(* CoDeSys 2.3.9.28 project: VISUALIZACIONBOTELLAS.pro *)
(* Libraries: Standard.lib 4.10.05 13:14:46, IecSfc.lib 13.4.06 16:51:28, SYSLIBCALLBACK.LIB 26.9.08 17:43:52 *)

(* Global variable list: Global_Variables *)
VAR_GLOBAL
   MATRIZ: ARRAY [1..5,1..10] OF REAL:=10(0),10(0),10(0),10(0),10(0);
   TIPO: ARRAY [1..10] OF INT:=1,2,2,1,1,2,2,1,1,2;
   C1:BOOL;
   C2:BOOL;
  C3:BOOL;
  C4:BOOL;
   AG:BOOL;
   LLENAR_AGUA:BOOL;
   ETIQUETAR:BOOL;
   NIVELAGUA:REAL;
   LTH:BOOL;
   LTL:BOOL;
   S2:BOOL;
   S3:BOOL;
   S4:BOOL;
  S5:BOOL;
  S6:BOOL;
   S7:BOOL;
   S8:BOOL;
   Sup1:BOOL;
   Inf1:BOOL;
	Sup2:BOOL;
   Inf2:BOOL;
   TIPO1:BOOL;
   TIPO2:BOOL;
   LLENAR:BOOL;
   LLENARTANQUE:BOOL;
   ESTIRATAP1:BOOL;
   RETRAETAP1:BOOL;
	PISTONC3:REAL;
	ESTIRATAP2:BOOL;
   RETRAETAP2:BOOL;
	PISTONC4:REAL;
   TAPONAR1:BOOL;
   TAPONAR2:BOOL;
   (*botones*)
   BOTONC1:BOOL;
   BOTONC2:BOOL;
	BOTONC3:BOOL;
   BOTONC4:BOOL;
   BOTONLLENAR:BOOL;
   BOTONLLENARTANQUE:BOOL;
  BOTONAG:BOOL;
 BOTONESTIRAPISTON3:BOOL;
	BOTONRETRAEPISTON3:BOOL;
	BOTONESTIRAPISTON4:BOOL;
	BOTONRETRAEPISTON4:BOOL;
	BOTONTAPONAR1:BOOL;
	BOTONTAPONAR2:BOOL;
(*VARIABLES MODO OPERACIÓN*)
    MANUAL:BOOL;
    AUTO:BOOL;
    C2OCUP:BOOL;
    TANQUELLENANDO:BOOL;
    TANQUEVACIO:BOOL;
    M:BOOL;
    PARO:BOOL;
    MARCHA:BOOL;
    MODORESET:BOOL;
(*variables temporizadores*)
    AT2:BOOL;
    FT2:BOOL;
    AT1:BOOL;
    FT1:BOOL;
    AT3:BOOL;
    FT3:BOOL;
  	AT4:BOOL;
    FT4:BOOL;
    Vectorcola:ARRAY [1..11] OF INT;
    ACCOMPLISHED:BOOL;
	TAPONADORA2OCU:BOOL;
    TAPONADORA1OCU:BOOL;
    RESETC3:BOOL;
    RESETC4:BOOL;
(*variables creadas*)
	C2OCU: BOOL;
	DEPOSOCU: BOOL;
	FLANCOS2SUBIDA: BOOL;
	FLANCOS4SUBIDA: BOOL;
	FLANCOS5SUBIDA: BOOL;
	FLANCOS7BAJADA: BOOL;
	FLANCOS34BAJADA: BOOL;
	FLANCOS8BAJADA: BOOL;
	TAP1OCU: BOOL;
	TAP2OCU: BOOL;
	CONTROLTANQUE: BOOL;
	AT30: BOOL;
	FT30: BOOL;

END_VAR

(* POU PLC_PRG, ST *)
PROGRAM PLC_PRG
VAR
END_VAR
VISUALIZACION;
MODOS;
TEMPOYCONTA;
END_PROGRAM

(* POU VISUALIZACION, ST *)
PROGRAM VISUALIZACION
VAR
	T1:TON;
	TH_OUT: BOOL;
    I:INT;
	RETRAETAP1THEN: BOOL;
END_VAR
AUTO:=NOT MANUAL;

T1(IN:=C1 AND NOT TH_OUT,PT:=T#4s,Q=>TH_OUT);
(*HACER VISIBLES BOTELLAS*)

IF C1=TRUE AND TH_OUT=TRUE AND MODORESET=FALSE THEN
   FOR I:=1 TO 10 BY 1 DO
      IF MATRIZ[1,I]=0 THEN
        MATRIZ[1,I]:=1;
        EXIT;
	  END_IF;
   END_FOR;
END_IF;

(*MOVIMIENTO BOTELLAS, PRIMER TRAMO HASTA 590*)
FOR I:=1 TO 10 BY 1 DO
   IF C1=TRUE AND MATRIZ[1,I]=1 AND MATRIZ[2,I]<590  THEN
     IF MODORESET=FALSE THEN
      MATRIZ[2,I]:=MATRIZ[2,I]+2;
    ELSE
       IF MATRIZ[2,I]>1 THEN
            MATRIZ[2,I]:=MATRIZ[2,I]+2;
      END_IF;
    END_IF;
   END_IF;
END_FOR;

(*LLENAR BOTELLAS*)

FOR I:=1 TO 10 BY 1 DO
	IF MATRIZ[2,I]>419 AND MATRIZ[2,I]<431 AND LLENAR=TRUE AND MATRIZ[5,I]=0 THEN
  	 MATRIZ[5,I]:=1;
	EXIT;
	END_IF;
END_FOR;
(*MOVIMIENTO EN LA SEGUNDA CINTA*)
FOR I:=1 TO 10 BY 1 DO
   IF C2=TRUE AND MATRIZ[1,I]=1 AND MATRIZ[2,I]>=575 AND MATRIZ[2,I]<730 AND AG=1 THEN
      MATRIZ[2,I]:=MATRIZ[2,I]+4;
      MATRIZ[3,I]:=MATRIZ[3,I]-4;
       IF MATRIZ[3,I]<=-130 THEN

         MATRIZ[3,I]:=-130;
       END_IF;
   END_IF;
IF C2=TRUE AND MATRIZ[1,I]=1 AND MATRIZ[2,I]>=575 AND MATRIZ[2,I]<734  AND AG=0 THEN
      MATRIZ[2,I]:=MATRIZ[2,I]+4;
      MATRIZ[3,I]:=MATRIZ[3,I]+4;
       IF MATRIZ[3,I]>=140 THEN
           MATRIZ[3,I]:=140;
      END_IF;
   END_IF;
END_FOR;

(*CINTA3*)
FOR I:=1 TO 10 BY 1 DO
   IF C3=TRUE AND MATRIZ[1,I]=1 AND MATRIZ[2,I]>=730 AND MATRIZ[3,I]<0 THEN
        MATRIZ[2,I]:=MATRIZ[2,I]+2;

       END_IF;
END_FOR;

(*CINTA3*)
FOR I:=1 TO 10 BY 1 DO
   IF C4=TRUE AND MATRIZ[1,I]=1 AND MATRIZ[2,I]>=730 AND MATRIZ[3,I]>0 THEN
        MATRIZ[2,I]:=MATRIZ[2,I]+2;
   END_IF;
END_FOR;

(*TANQUE*)
IF LLENAR=TRUE THEN
 NIVELAGUA:=NIVELAGUA+1;
 IF NIVELAGUA>198 THEN
     NIVELAGUA:=198;
 END_IF;
END_IF

IF LLENARTANQUE=TRUE THEN
 NIVELAGUA:=NIVELAGUA-2;
 IF NIVELAGUA<=0 THEN
     NIVELAGUA:=0;
 END_IF;
END_IF

(*PISTON TAPONADORA 1*)
IF ESTIRATAP1 THEN
PISTONC3:=PISTONC3+3;
      IF PISTONC3>=+30 THEN
           PISTONC3:=+30;
     END_IF;

END_IF;
IF RETRAETAP1 THEN
      PISTONC3:=PISTONC3-3;
      IF PISTONC3<=0 THEN
           PISTONC3:=0;
     END_IF;
END_IF;

(*PISTON TAPONADORA 2*)
IF ESTIRATAP2 THEN
PISTONC4:=PISTONC4+3;
      IF PISTONC4>=+40 THEN
           PISTONC4:=+40;
     END_IF;

END_IF;
IF RETRAETAP2 THEN
      PISTONC4:=PISTONC4-3;
      IF PISTONC4<=0 THEN
           PISTONC4:=0;
     END_IF;
END_IF;

(*SENSORES*)
FOR I:=1 TO 10 BY 1 DO
   IF MATRIZ[2,I]>419 AND MATRIZ[2,I]<431 AND TIPO[I]=1 THEN
         TIPO1:=TRUE;
         EXIT;
   ELSE
         TIPO1:=FALSE;
   END_IF;
   IF MATRIZ[2,I]>419 AND MATRIZ[2,I]<431 AND TIPO[I]=2 THEN
         TIPO2:=TRUE;
         EXIT;
   ELSE
         TIPO2:=FALSE;
   END_IF;
END_FOR;


FOR I:=1 TO 10 BY 1 DO
   IF MATRIZ[2,I]>570 AND MATRIZ[2,I]<600 THEN
         S2:=TRUE;
         EXIT;
   ELSE
         S2:=FALSE;
   END_IF;
END_FOR;

IF NIVELAGUA<2 THEN
    LTH:=TRUE;
ELSE
    LTH:=FALSE;
END_IF;

IF NIVELAGUA<90 THEN
    LTL:=TRUE;
ELSE
    LTL:=FALSE;
END_IF;

FOR I:=1 TO 10 BY 1 DO
   IF MATRIZ[2,I]>733 AND MATRIZ[2,I]<745 AND MATRIZ[3,I]>0 THEN
         S3:=TRUE;
         EXIT;
   ELSE
         S3:=FALSE;
   END_IF;
END_FOR;


FOR I:=1 TO 10 BY 1 DO
   IF MATRIZ[2,I]>729 AND MATRIZ[2,I]<745 AND MATRIZ[3,I] <0 THEN
         S4:=TRUE;
         EXIT;
   ELSE
         S4:=FALSE;
   END_IF;
END_FOR;

FOR I:=1 TO 10 BY 1 DO
   IF MATRIZ[2,I]>920 AND MATRIZ[2,I]<935 AND MATRIZ[3,I] <0 THEN
         S6:=TRUE;
         EXIT;
   ELSE
         S6:=FALSE;
   END_IF;
END_FOR;

FOR I:=1 TO 10 BY 1 DO
   IF MATRIZ[2,I]>1075 AND MATRIZ[2,I]<1090 AND MATRIZ[3,I] <0 THEN
         S8:=TRUE;
         EXIT;
   ELSE
         S8:=FALSE;
   END_IF;
END_FOR;


FOR I:=1 TO 10 BY 1 DO
   IF MATRIZ[2,I]>920 AND MATRIZ[2,I]<935 AND MATRIZ[3,I] >0 THEN
         S5:=TRUE;
         EXIT;
   ELSE
         S5:=FALSE;
   END_IF;
END_FOR;

FOR I:=1 TO 10 BY 1 DO
   IF MATRIZ[2,I]>1075 AND MATRIZ[2,I]<1090 AND MATRIZ[3,I] >0 THEN
         S7:=TRUE;
         EXIT;
   ELSE
         S7:=FALSE;
   END_IF;
END_FOR;
(*PISTON C3*)
IF PISTONC3=0 THEN
     Sup1:=TRUE;
ELSE
    Sup1:=FALSE;
END_IF;
IF PISTONC3>29 THEN
     Inf1:=TRUE;
ELSE
    Inf1:=FALSE;
END_IF;

(*PISTON C4*)
IF PISTONC4=0 THEN
     Sup2:=TRUE;
ELSE
    Sup2:=FALSE;
END_IF;
IF PISTONC4>39 THEN
     Inf2:=TRUE;
ELSE
    Inf2:=FALSE;
END_IF;


(*REINICIO DE TODO*)

FOR I:=1 TO 10 BY 1 DO
   IF MATRIZ[2,I]>=1089  THEN
    MATRIZ[1,I]:=0;
    MATRIZ[2,I]:=0;
    MATRIZ[3,I]:=0;
   MATRIZ[4,I]:=0;
   MATRIZ[5,I]:=0;
   END_IF;
END_FOR;
END_PROGRAM

(* POU MODOS, SFC *)
PROGRAM MODOS
VAR
	AUTOMATICO: BOOL;
END_VAR
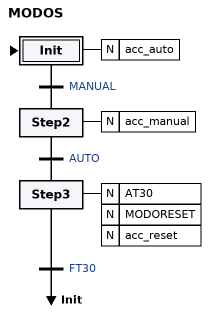
INITIAL_STEP Init:
	acc_auto(N);
END_STEP
TRANSITION FROM Init TO Step2 := MANUAL;
END_TRANSITION
STEP Step2:
	acc_manual(N);
END_STEP
TRANSITION FROM Step2 TO Step3 := AUTO;
END_TRANSITION
STEP Step3:
	AT30(N);
	MODORESET(N);
	acc_reset(N);
END_STEP
TRANSITION FROM Step3 TO Init := FT30;
END_TRANSITION
END_PROGRAM
ACTION acc_auto:
AUTOMATICO1;
END_ACTION
ACTION acc_manual:
MANUAL_PROG;
END_ACTION
ACTION acc_reset:
REINICIO;
Encolar;
Mover_cinta2;
END_ACTION

(* POU AUTOMATICO1, SFC *)
PROGRAM AUTOMATICO1
VAR
END_VAR
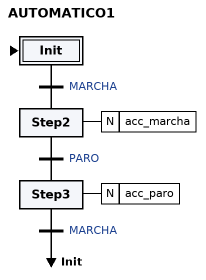
INITIAL_STEP Init:
END_STEP
TRANSITION FROM Init TO Step2 := MARCHA;
END_TRANSITION
STEP Step2:
	acc_marcha(N);
END_STEP
TRANSITION FROM Step2 TO Step3 := PARO;
END_TRANSITION
STEP Step3:
	acc_paro(N);
END_STEP
TRANSITION FROM Step3 TO Init := MARCHA;
END_TRANSITION
END_PROGRAM
ACTION acc_marcha:
Cinta1;
CINTA2;
CINTA3;
CINTA4;
Tanque1;
TANQUE2;
TAPONADOR1;
TAPONADOR2;
Encolar;
Mover_cinta2;
END_ACTION
ACTION acc_paro:
PARO1;
Tanque1;
TAPONADOR1;
TAPONADOR2;
END_ACTION

(* POU Cinta1, LD *)
PROGRAM Cinta1
VAR
END_VAR
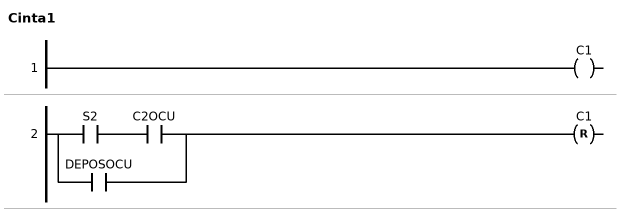
_LD_ (* Ladder Diagram *)
NETWORK 1
	* --- (C1)
NETWORK 2
	{ [S2] - [C2OCU] | [DEPOSOCU] } --- (R C1)
_END_LD_
(* the same logic as Structured Text *)
(* Network 1 *)
C1 := TRUE;
(* Network 2 *)
IF S2 AND C2OCU OR DEPOSOCU THEN C1 := FALSE; END_IF;
END_PROGRAM

(* POU PARO1, LD *)
PROGRAM PARO1
VAR
END_VAR
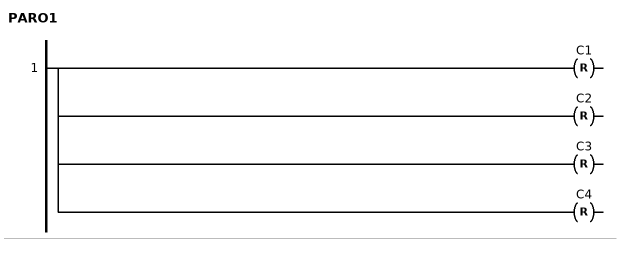
_LD_ (* Ladder Diagram *)
NETWORK 1
	* --- (R C1) (R C2) (R C3) (R C4)
_END_LD_
(* the same logic as Structured Text *)
(* Network 1 *)
C1 := FALSE;
C2 := FALSE;
C3 := FALSE;
C4 := FALSE;
END_PROGRAM

(* POU MANUAL_PROG, LD *)
PROGRAM MANUAL_PROG
VAR
END_VAR
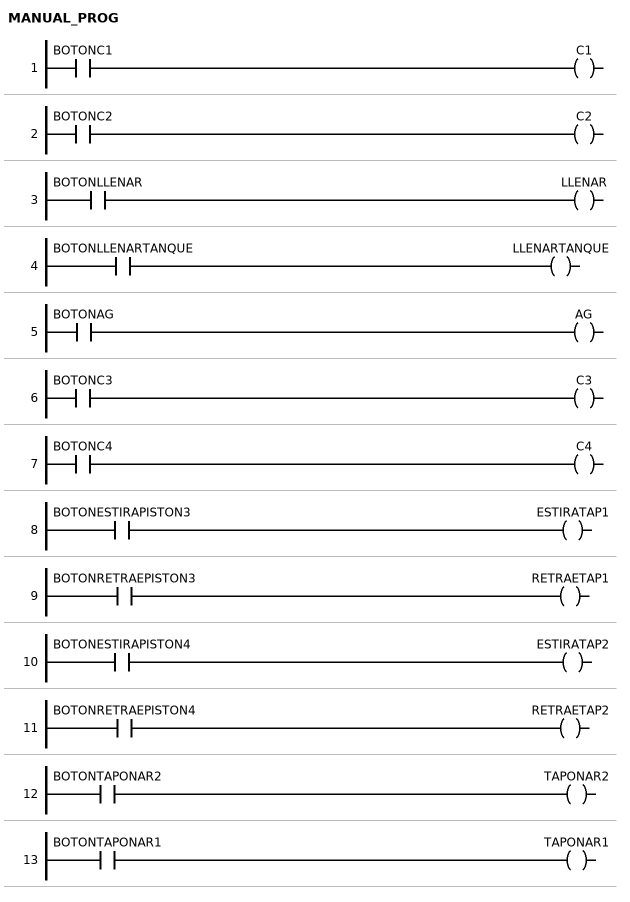
_LD_ (* Ladder Diagram *)
NETWORK 1
	[BOTONC1] --- (C1)
NETWORK 2
	[BOTONC2] --- (C2)
NETWORK 3
	[BOTONLLENAR] --- (LLENAR)
NETWORK 4
	[BOTONLLENARTANQUE] --- (LLENARTANQUE)
NETWORK 5
	[BOTONAG] --- (AG)
NETWORK 6
	[BOTONC3] --- (C3)
NETWORK 7
	[BOTONC4] --- (C4)
NETWORK 8
	[BOTONESTIRAPISTON3] --- (ESTIRATAP1)
NETWORK 9
	[BOTONRETRAEPISTON3] --- (RETRAETAP1)
NETWORK 10
	[BOTONESTIRAPISTON4] --- (ESTIRATAP2)
NETWORK 11
	[BOTONRETRAEPISTON4] --- (RETRAETAP2)
NETWORK 12
	[BOTONTAPONAR2] --- (TAPONAR2)
NETWORK 13
	[BOTONTAPONAR1] --- (TAPONAR1)
_END_LD_
(* the same logic as Structured Text *)
(* Network 1 *)
C1 := BOTONC1;
(* Network 2 *)
C2 := BOTONC2;
(* Network 3 *)
LLENAR := BOTONLLENAR;
(* Network 4 *)
LLENARTANQUE := BOTONLLENARTANQUE;
(* Network 5 *)
AG := BOTONAG;
(* Network 6 *)
C3 := BOTONC3;
(* Network 7 *)
C4 := BOTONC4;
(* Network 8 *)
ESTIRATAP1 := BOTONESTIRAPISTON3;
(* Network 9 *)
RETRAETAP1 := BOTONRETRAEPISTON3;
(* Network 10 *)
ESTIRATAP2 := BOTONESTIRAPISTON4;
(* Network 11 *)
RETRAETAP2 := BOTONRETRAEPISTON4;
(* Network 12 *)
TAPONAR2 := BOTONTAPONAR2;
(* Network 13 *)
TAPONAR1 := BOTONTAPONAR1;
END_PROGRAM

(* POU REINICIO, LD *)
PROGRAM REINICIO
VAR
END_VAR
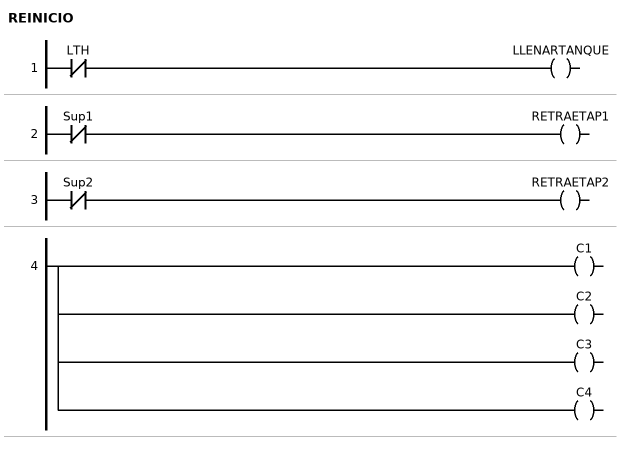
_LD_ (* Ladder Diagram *)
NETWORK 1
	[/LTH] --- (LLENARTANQUE)
NETWORK 2
	[/Sup1] --- (RETRAETAP1)
NETWORK 3
	[/Sup2] --- (RETRAETAP2)
NETWORK 4
	* --- (C1) (C2) (C3) (C4)
_END_LD_
(* the same logic as Structured Text *)
(* Network 1 *)
LLENARTANQUE := NOT LTH;
(* Network 2 *)
RETRAETAP1 := NOT Sup1;
(* Network 3 *)
RETRAETAP2 := NOT Sup2;
(* Network 4 *)
C1 := TRUE;
C2 := TRUE;
C3 := TRUE;
C4 := TRUE;
END_PROGRAM

(* POU TEMPOYCONTA, LD *)
PROGRAM TEMPOYCONTA
VAR
	T1: TON;
	T2: TON;
	T3: TON;
	T4: TON;
	T30: TON;


END_VAR
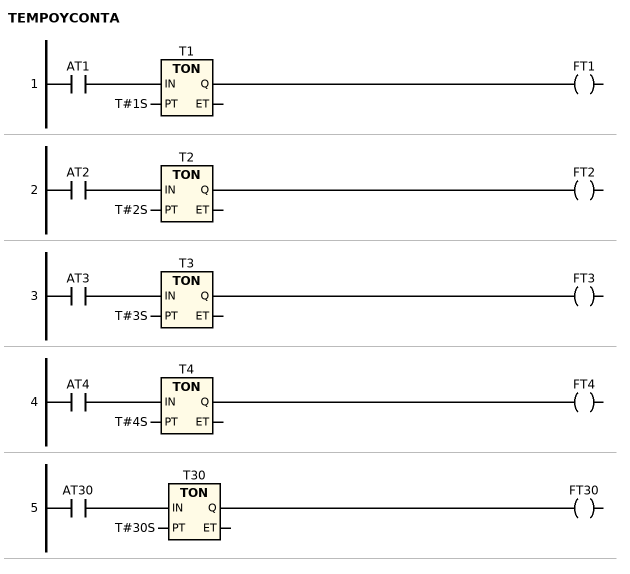
_LD_ (* Ladder Diagram *)
NETWORK 1
	[AT1] - T1:TON(IN: *, PT: T#1S) --- (FT1)
NETWORK 2
	[AT2] - T2:TON(IN: *, PT: T#2S) --- (FT2)
NETWORK 3
	[AT3] - T3:TON(IN: *, PT: T#3S) --- (FT3)
NETWORK 4
	[AT4] - T4:TON(IN: *, PT: T#4S) --- (FT4)
NETWORK 5
	[AT30] - T30:TON(IN: *, PT: T#30S) --- (FT30)
_END_LD_
(* the same logic as Structured Text *)
(* Network 1 *)
T1(IN := AT1, PT := T#1S);
FT1 := T1.Q;
(* Network 2 *)
T2(IN := AT2, PT := T#2S);
FT2 := T2.Q;
(* Network 3 *)
T3(IN := AT3, PT := T#3S);
FT3 := T3.Q;
(* Network 4 *)
T4(IN := AT4, PT := T#4S);
FT4 := T4.Q;
(* Network 5 *)
T30(IN := AT30, PT := T#30S);
FT30 := T30.Q;
END_PROGRAM

(* POU CINTA2, LD *)
PROGRAM CINTA2
VAR
	TRIG1: R_TRIG;
	TRIG2: F_TRIG;
	TRIG3: F_TRIG;
	CTUD1: CTUD;
	RESETC2: BOOL;

END_VAR
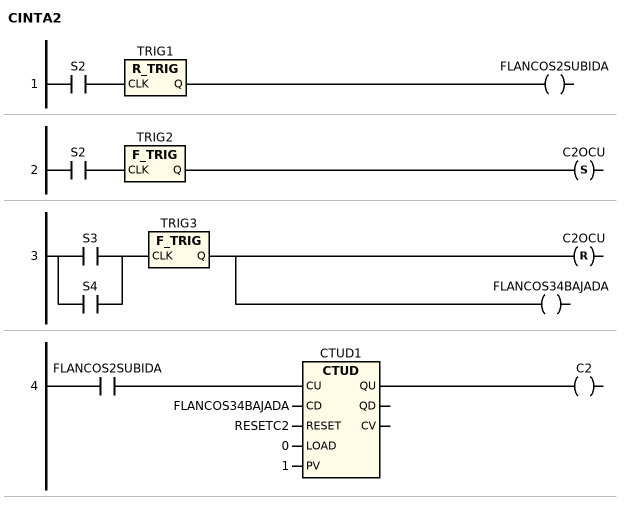
_LD_ (* Ladder Diagram *)
NETWORK 1
	[S2] - TRIG1:R_TRIG(CLK: *) --- (FLANCOS2SUBIDA)
NETWORK 2
	[S2] - TRIG2:F_TRIG(CLK: *) --- (S C2OCU)
NETWORK 3
	{ [S3] | [S4] } - TRIG3:F_TRIG(CLK: *) --- (R C2OCU) (FLANCOS34BAJADA)
NETWORK 4
	[FLANCOS2SUBIDA] - CTUD1:CTUD(CU: *, CD: FLANCOS34BAJADA, RESET: RESETC2, LOAD: 0, PV: 1) --- (C2)
_END_LD_
(* the same logic as Structured Text *)
(* Network 1 *)
TRIG1(CLK := S2);
FLANCOS2SUBIDA := TRIG1.Q;
(* Network 2 *)
TRIG2(CLK := S2);
IF TRIG2.Q THEN C2OCU := TRUE; END_IF;
(* Network 3 *)
TRIG3(CLK := S3 OR S4);
IF TRIG3.Q THEN C2OCU := FALSE; END_IF;
FLANCOS34BAJADA := TRIG3.Q;
(* Network 4 *)
CTUD1(CU := FLANCOS2SUBIDA, CD := FLANCOS34BAJADA, RESET := RESETC2, LOAD := 0, PV := 1);
C2 := CTUD1.QU;
END_PROGRAM

(* POU CINTA3, LD *)
PROGRAM CINTA3
VAR
	TRIG1: R_TRIG;
	TRIG2: F_TRIG;
    CTUD1:  CTUD;
END_VAR
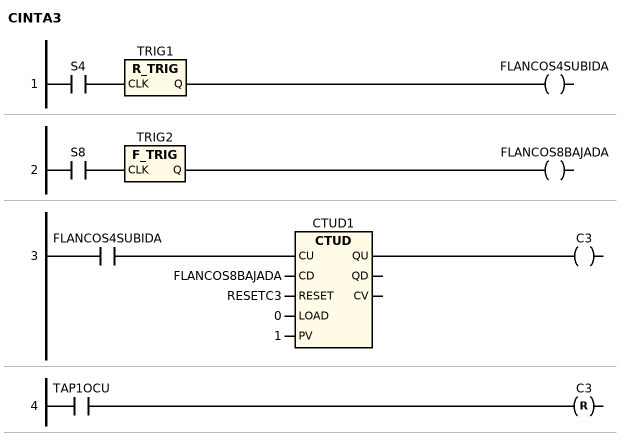
_LD_ (* Ladder Diagram *)
NETWORK 1
	[S4] - TRIG1:R_TRIG(CLK: *) --- (FLANCOS4SUBIDA)
NETWORK 2
	[S8] - TRIG2:F_TRIG(CLK: *) --- (FLANCOS8BAJADA)
NETWORK 3
	[FLANCOS4SUBIDA] - CTUD1:CTUD(CU: *, CD: FLANCOS8BAJADA, RESET: RESETC3, LOAD: 0, PV: 1) --- (C3)
NETWORK 4
	[TAP1OCU] --- (R C3)
_END_LD_
(* the same logic as Structured Text *)
(* Network 1 *)
TRIG1(CLK := S4);
FLANCOS4SUBIDA := TRIG1.Q;
(* Network 2 *)
TRIG2(CLK := S8);
FLANCOS8BAJADA := TRIG2.Q;
(* Network 3 *)
CTUD1(CU := FLANCOS4SUBIDA, CD := FLANCOS8BAJADA, RESET := RESETC3, LOAD := 0, PV := 1);
C3 := CTUD1.QU;
(* Network 4 *)
IF TAP1OCU THEN C3 := FALSE; END_IF;
END_PROGRAM

(* POU CINTA4, LD *)
PROGRAM CINTA4
VAR
	TRIG1: R_TRIG;
	TRIG2: F_TRIG;
    CTUD1:  CTUD;
END_VAR
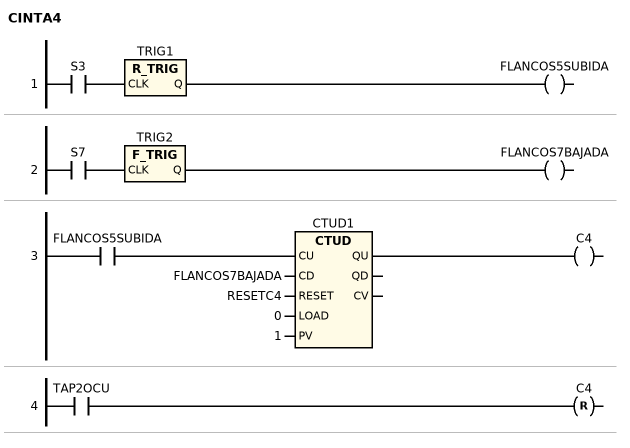
_LD_ (* Ladder Diagram *)
NETWORK 1
	[S3] - TRIG1:R_TRIG(CLK: *) --- (FLANCOS5SUBIDA)
NETWORK 2
	[S7] - TRIG2:F_TRIG(CLK: *) --- (FLANCOS7BAJADA)
NETWORK 3
	[FLANCOS5SUBIDA] - CTUD1:CTUD(CU: *, CD: FLANCOS7BAJADA, RESET: RESETC4, LOAD: 0, PV: 1) --- (C4)
NETWORK 4
	[TAP2OCU] --- (R C4)
_END_LD_
(* the same logic as Structured Text *)
(* Network 1 *)
TRIG1(CLK := S3);
FLANCOS5SUBIDA := TRIG1.Q;
(* Network 2 *)
TRIG2(CLK := S7);
FLANCOS7BAJADA := TRIG2.Q;
(* Network 3 *)
CTUD1(CU := FLANCOS5SUBIDA, CD := FLANCOS7BAJADA, RESET := RESETC4, LOAD := 0, PV := 1);
C4 := CTUD1.QU;
(* Network 4 *)
IF TAP2OCU THEN C4 := FALSE; END_IF;
END_PROGRAM

(* POU Encolar, ST *)
PROGRAM Encolar
VAR


	TIPO1a:BOOL;
    TIPO2a:BOOL;


	I: INT;

	Acca: BOOL;

END_VAR
IF TIPO1=TRUE AND TIPO1a=FALSE THEN
	FOR I:= 1 TO 10 BY 1 DO
		IF Vectorcola[I] = 0 THEN
			Vectorcola[I]:= 1;
			EXIT;
		END_IF;
	END_FOR;
END_IF;


IF TIPO2=TRUE AND TIPO2a=FALSE THEN
	FOR I:= 1 TO 10 BY 1 DO
		IF Vectorcola[I] = 0 THEN
			Vectorcola[I]:= 2;
			EXIT;
		END_IF;
	END_FOR;
END_IF;


IF ACCOMPLISHED = TRUE AND ACCa = FALSE THEN
	FOR I:=1 TO 10 BY 1 DO
		Vectorcola[I]:= Vectorcola[I+1];
	END_FOR;
		Vectorcola[10]:= 0;
	END_IF;




TIPO1a:=TIPO1;
TIPO2a:=TIPO2;
Acca:= ACCOMPLISHED;
END_PROGRAM

(* POU Mover_cinta2, SFC *)
PROGRAM Mover_cinta2
VAR
END_VAR
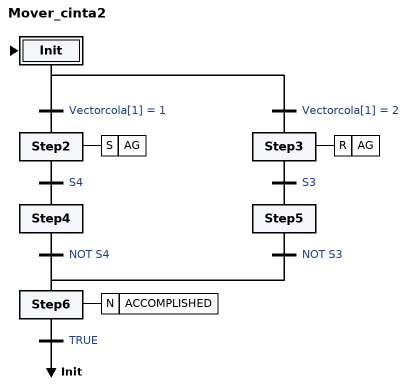
INITIAL_STEP Init:
END_STEP
TRANSITION FROM Init TO Step2 := Vectorcola[1] = 1;
END_TRANSITION
TRANSITION FROM Init TO Step3 := Vectorcola[1] = 2;
END_TRANSITION
STEP Step2:
	AG(S);
END_STEP
TRANSITION FROM Step2 TO Step4 := S4;
END_TRANSITION
STEP Step4:
END_STEP
TRANSITION FROM Step4 TO Step6 := NOT S4;
END_TRANSITION
STEP Step3:
	AG(R);
END_STEP
TRANSITION FROM Step3 TO Step5 := S3;
END_TRANSITION
STEP Step5:
END_STEP
TRANSITION FROM Step5 TO Step6 := NOT S3;
END_TRANSITION
STEP Step6:
	ACCOMPLISHED(N);
END_STEP
TRANSITION FROM Step6 TO Init := TRUE;
END_TRANSITION
END_PROGRAM

(* POU Tanque1, SFC *)
PROGRAM Tanque1
VAR
END_VAR
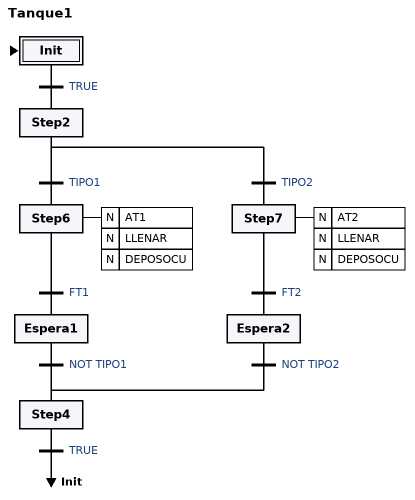
INITIAL_STEP Init:
END_STEP
TRANSITION FROM Init TO Step2 := TRUE;
END_TRANSITION
STEP Step2:
END_STEP
TRANSITION FROM Step2 TO Step6 := TIPO1;
END_TRANSITION
TRANSITION FROM Step2 TO Step7 := TIPO2;
END_TRANSITION
STEP Step6:
	AT1(N);
	LLENAR(N);
	DEPOSOCU(N);
END_STEP
TRANSITION FROM Step6 TO Espera1 := FT1;
END_TRANSITION
STEP Espera1:
END_STEP
TRANSITION FROM Espera1 TO Step4 := NOT TIPO1;
END_TRANSITION
STEP Step7:
	AT2(N);
	LLENAR(N);
	DEPOSOCU(N);
END_STEP
TRANSITION FROM Step7 TO Espera2 := FT2;
END_TRANSITION
STEP Espera2:
END_STEP
TRANSITION FROM Espera2 TO Step4 := NOT TIPO2;
END_TRANSITION
STEP Step4:
END_STEP
TRANSITION FROM Step4 TO Init := TRUE;
END_TRANSITION
END_PROGRAM

(* POU TANQUE2, LD *)
PROGRAM TANQUE2
VAR
END_VAR
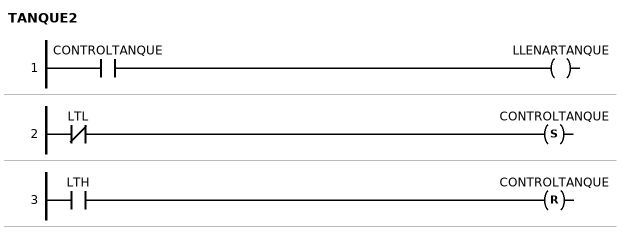
_LD_ (* Ladder Diagram *)
NETWORK 1
	[CONTROLTANQUE] --- (LLENARTANQUE)
NETWORK 2
	[/LTL] --- (S CONTROLTANQUE)
NETWORK 3
	[LTH] --- (R CONTROLTANQUE)
_END_LD_
(* the same logic as Structured Text *)
(* Network 1 *)
LLENARTANQUE := CONTROLTANQUE;
(* Network 2 *)
IF NOT LTL THEN CONTROLTANQUE := TRUE; END_IF;
(* Network 3 *)
IF LTH THEN CONTROLTANQUE := FALSE; END_IF;
END_PROGRAM

(* POU TAPONADOR1, SFC *)
PROGRAM TAPONADOR1
VAR
END_VAR
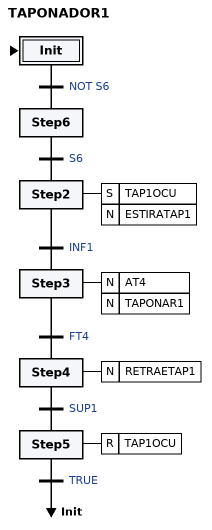
INITIAL_STEP Init:
END_STEP
TRANSITION FROM Init TO Step6 := NOT S6;
END_TRANSITION
STEP Step6:
END_STEP
TRANSITION FROM Step6 TO Step2 := S6;
END_TRANSITION
STEP Step2:
	TAP1OCU(S);
	ESTIRATAP1(N);
END_STEP
TRANSITION FROM Step2 TO Step3 := INF1;
END_TRANSITION
STEP Step3:
	AT4(N);
	TAPONAR1(N);
END_STEP
TRANSITION FROM Step3 TO Step4 := FT4;
END_TRANSITION
STEP Step4:
	RETRAETAP1(N);
END_STEP
TRANSITION FROM Step4 TO Step5 := SUP1;
END_TRANSITION
STEP Step5:
	TAP1OCU(R);
END_STEP
TRANSITION FROM Step5 TO Init := TRUE;
END_TRANSITION
END_PROGRAM

(* POU TAPONADOR2, SFC *)
PROGRAM TAPONADOR2
VAR
END_VAR
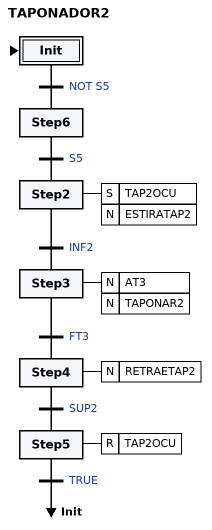
INITIAL_STEP Init:
END_STEP
TRANSITION FROM Init TO Step6 := NOT S5;
END_TRANSITION
STEP Step6:
END_STEP
TRANSITION FROM Step6 TO Step2 := S5;
END_TRANSITION
STEP Step2:
	TAP2OCU(S);
	ESTIRATAP2(N);
END_STEP
TRANSITION FROM Step2 TO Step3 := INF2;
END_TRANSITION
STEP Step3:
	AT3(N);
	TAPONAR2(N);
END_STEP
TRANSITION FROM Step3 TO Step4 := FT3;
END_TRANSITION
STEP Step4:
	RETRAETAP2(N);
END_STEP
TRANSITION FROM Step4 TO Step5 := SUP2;
END_TRANSITION
STEP Step5:
	TAP2OCU(R);
END_STEP
TRANSITION FROM Step5 TO Init := TRUE;
END_TRANSITION
END_PROGRAM

(* Visualisation VISUAL
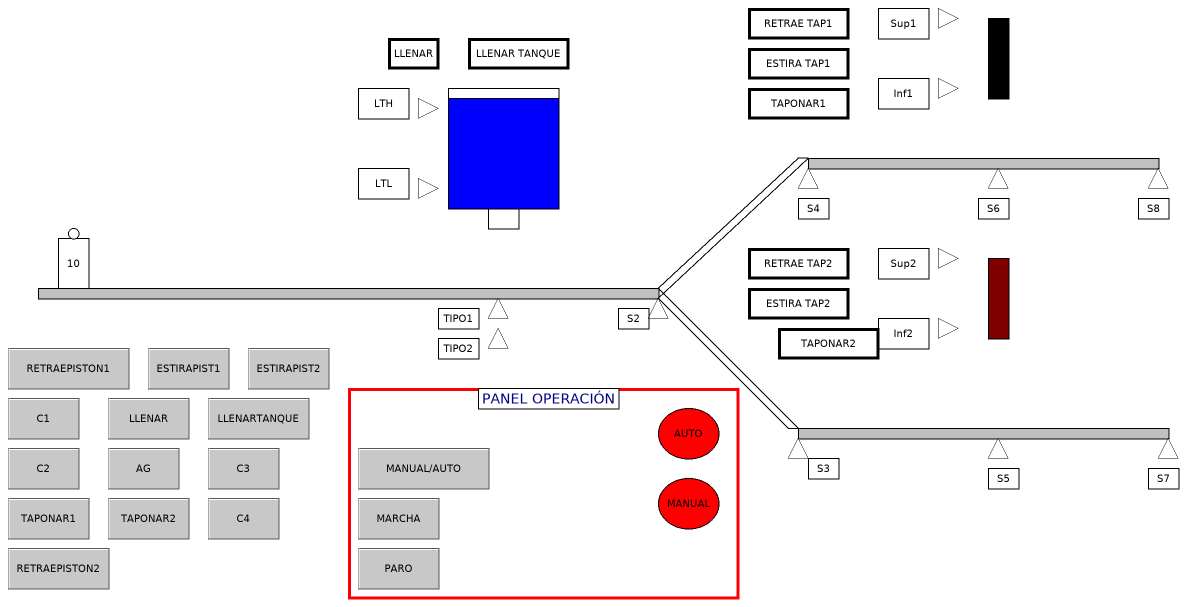
rectangle at (60,260)-(91,291): text "1"; invisible if MATRIZ[1,1]=0; alarm colour if MATRIZ[5,1]; x offset MATRIZ[2,1]; y offset MATRIZ[3,1]
ellipse at (70,250)-(81,261): invisible if MATRIZ[1,1]=0; x offset MATRIZ[2,1]; y offset MATRIZ[3,1]
rectangle at (60,240)-(91,291): text "2"; invisible if MATRIZ[1,2]=0; alarm colour if MATRIZ[5,2]; x offset MATRIZ[2,2]; y offset MATRIZ[3,2]
ellipse at (70,230)-(81,241): invisible if MATRIZ[1,2]=0; x offset MATRIZ[2,2]; y offset MATRIZ[3,2]
rectangle at (60,240)-(91,291): text "3"; invisible if MATRIZ[1,3]=0; alarm colour if MATRIZ[5,3]; x offset MATRIZ[2,3]; y offset MATRIZ[3,3]
ellipse at (70,230)-(81,241): invisible if MATRIZ[1,3]=0; x offset MATRIZ[2,3]; y offset MATRIZ[3,3]
rectangle at (60,260)-(91,291): text "4"; invisible if MATRIZ[1,4]=0; alarm colour if MATRIZ[5,4]; x offset MATRIZ[2,4]; y offset MATRIZ[3,4]
ellipse at (70,250)-(81,261): invisible if MATRIZ[1,4]=0; x offset MATRIZ[2,4]; y offset MATRIZ[3,4]
rectangle at (60,260)-(91,291): text "5"; invisible if MATRIZ[1,5]=0; alarm colour if MATRIZ[5,5]; x offset MATRIZ[2,5]; y offset MATRIZ[3,5]
ellipse at (70,250)-(81,261): invisible if MATRIZ[1,5]=0; x offset MATRIZ[2,5]; y offset MATRIZ[3,5]
rectangle at (60,240)-(91,291): text "6"; invisible if MATRIZ[1,6]=0; alarm colour if MATRIZ[5,6]; x offset MATRIZ[2,6]; y offset MATRIZ[3,6]
ellipse at (70,230)-(81,241): invisible if MATRIZ[1,6]=0; x offset MATRIZ[2,6]; y offset MATRIZ[3,6]
rectangle at (60,240)-(91,291): text "7"; invisible if MATRIZ[1,7]=0; alarm colour if MATRIZ[5,7]; x offset MATRIZ[2,7]; y offset MATRIZ[3,7]
ellipse at (70,230)-(81,241): invisible if MATRIZ[1,7]=0; x offset MATRIZ[2,7]; y offset MATRIZ[3,7]
rectangle at (60,260)-(91,291): text "8"; invisible if MATRIZ[1,8]=0; alarm colour if MATRIZ[5,8]; x offset MATRIZ[2,8]; y offset MATRIZ[3,8]
ellipse at (70,250)-(81,261): invisible if MATRIZ[1,8]=0; x offset MATRIZ[2,8]; y offset MATRIZ[3,8]
rectangle at (60,260)-(91,291): text "9"; invisible if MATRIZ[1,9]=0; alarm colour if MATRIZ[5,9]; x offset MATRIZ[2,9]; y offset MATRIZ[3,9]
ellipse at (70,250)-(81,261): invisible if MATRIZ[1,9]=0; x offset MATRIZ[2,9]; y offset MATRIZ[2,9]
rectangle at (60,240)-(91,291): text "10"; invisible if MATRIZ[1,10]=0; alarm colour if MATRIZ[5,10]; x offset MATRIZ[2,10]; y offset MATRIZ[3,10]
ellipse at (70,230)-(81,241): invisible if MATRIZ[1,10]=0; x offset MATRIZ[2,10]; y offset MATRIZ[3,10]
rectangle at (40,290)-(661,301): alarm colour if C2
polygon at (490,300)-(510,320): alarm colour if TIPO1
polygon at (490,330)-(510,350): alarm colour if TIPO2
polygon at (650,300)-(670,320): alarm colour if S2
rectangle at (440,310)-(481,331): text "TIPO1"
rectangle at (440,340)-(481,361): text "TIPO2"
rectangle at (620,310)-(651,331): text "S2"
button at (10,400)-(81,441): text "C1"; toggles BOTONC1
rectangle at (490,210)-(521,231): alarm colour if LLENAR
polygon at (420,100)-(440,120): alarm colour if LTH
polygon at (420,180)-(440,200): alarm colour if LTL
rectangle at (360,90)-(411,121): text "LTH"
rectangle at (360,170)-(411,201): text "LTL"
rectangle at (450,100)-(561,211): top NIVELAGUA
button at (110,400)-(191,441): text "LLENAR"; taps BOTONLLENAR
button at (210,400)-(311,441): text "LLENARTANQUE"; taps BOTONLLENARTANQUE
rectangle at (390,40)-(441,71): text "LLENAR"; alarm colour if LLENAR
rectangle at (470,40)-(571,71): text "LLENAR TANQUE"; alarm colour if LLENARTANQUE
polyline at (660,160)-(810,300): invisible if AG=0; alarm colour if C2
polyline at (660,290)-(800,430): invisible if AG=1; alarm colour if C2
rectangle at (800,430)-(1171,441): alarm colour if C4
rectangle at (810,160)-(1161,171): alarm colour if C3
polygon at (790,440)-(810,460): alarm colour if S3
rectangle at (810,460)-(841,481): text "S3"
polygon at (800,170)-(820,190): alarm colour if S4
rectangle at (800,200)-(831,221): text "S4"
polygon at (990,170)-(1010,190): alarm colour if S6
polygon at (1150,170)-(1170,190): alarm colour if S8
polygon at (990,440)-(1010,460): alarm colour if S5
polygon at (1160,440)-(1180,460): alarm colour if S7
rectangle at (980,200)-(1011,221): text "S6"
rectangle at (1140,200)-(1171,221): text "S8"
rectangle at (990,470)-(1021,491): text "S5"
rectangle at (1150,470)-(1181,491): text "S7"
button at (10,450)-(81,491): text "C2"; toggles BOTONC2
button at (110,450)-(181,491): text "AG"; toggles BOTONAG
button at (210,450)-(281,491): text "C3"; toggles BOTONC3
button at (210,500)-(281,541): text "C4"; toggles BOTONC4
rectangle at (990,20)-(1011,101): bottom PISTONC3
polygon at (940,10)-(960,30): alarm colour if Sup1
polygon at (940,80)-(960,100): alarm colour if Inf1
rectangle at (880,10)-(931,41): text "Sup1"
rectangle at (880,80)-(931,111): text "Inf1"
button at (150,350)-(231,391): text "ESTIRAPIST1"; taps BOTONESTIRAPISTON3
button at (10,350)-(131,391): text "RETRAEPISTON1"; taps BOTONRETRAEPISTON3
rectangle at (750,10)-(851,41): text "RETRAE TAP1"; alarm colour if RETRAETAP1
rectangle at (750,50)-(851,81): text "ESTIRA TAP1"; alarm colour if ESTIRATAP1
rectangle at (990,260)-(1011,341): bottom PISTONC4
polygon at (940,250)-(960,270): alarm colour if Sup2
polygon at (940,320)-(960,340): alarm colour if Inf2
rectangle at (880,250)-(931,281): text "Sup2"
rectangle at (880,320)-(931,351): text "Inf2"
rectangle at (750,250)-(851,281): text "RETRAE TAP2"; alarm colour if RETRAETAP2
rectangle at (750,290)-(851,321): text "ESTIRA TAP2"; alarm colour if ESTIRATAP2
button at (250,350)-(331,391): text "ESTIRAPIST2"; taps BOTONESTIRAPISTON4
button at (10,550)-(111,591): text "RETRAEPISTON2"; taps BOTONRETRAEPISTON4
rectangle at (780,330)-(881,361): text "TAPONAR2"; alarm colour if TAPONAR2
rectangle at (750,90)-(851,121): text "TAPONAR1"; alarm colour if TAPONAR1
button at (10,500)-(91,541): text "TAPONAR1"; taps BOTONTAPONAR1
button at (110,500)-(191,541): text "TAPONAR2"; taps BOTONTAPONAR2
button at (360,450)-(491,491): text "MANUAL/AUTO"; toggles MANUAL
button at (360,500)-(441,541): text "MARCHA"; taps MARCHA
button at (360,550)-(441,591): text "PARO"; taps PARO
ellipse at (660,410)-(721,461): text "AUTO"; alarm colour if NOT MANUAL
ellipse at (660,480)-(721,531): text "MANUAL"; alarm colour if MANUAL
rectangle at (480,390)-(621,411): text "PANEL OPERACIÓN"
4 more shapes without text or variables
*)
